VAR_GLOBAL CONSTANT
	///ctrl commands definitions
	///specific commands >200 - every command has to be a even number
	cCMD_CLEAR: INT := 202;
END_VAR

(* stored: Version 1.1.0.1, ProductVersion 3.1.0.19
   GVL DPJ_CmdState: Id {a0ded7c9-ebd8-42ad-afdc-c20b3fec0fec} *)
